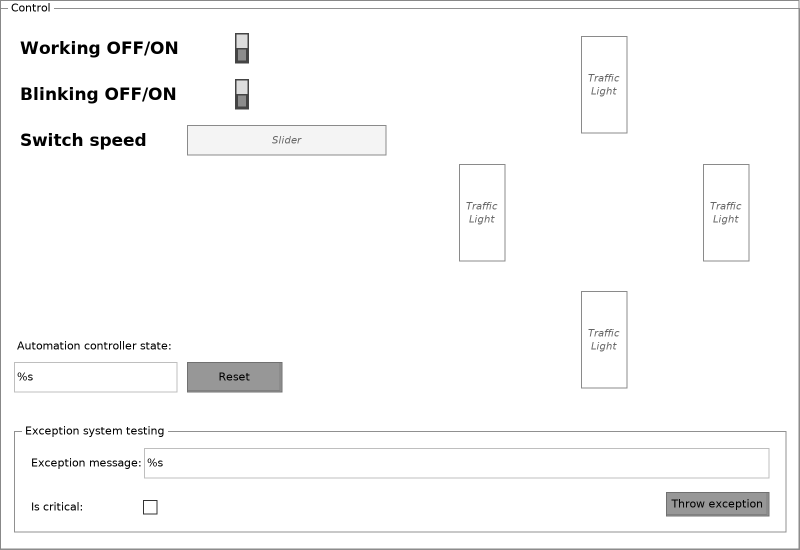
VISUALIZATION Intersection  // 800x550
    GroupBox (0,0 800x550), "Control"
        Label (17,33 166x30), "Working OFF/ON"
        Label (17,79 166x30), "Blinking OFF/ON"
        Rectangle (543,32 120x360), angle 90
        Line (486,126)
        Rectangle (543,24 120x376)
        Frame (581,36 46x97)
            shows TrafficLight(Red := Terminals.DO_2.Channel_4, Yellow := Terminals.DO_2.Channel_5, Green := Terminals.DO_2.Channel_6)
        Frame (581,291 46x97)
            shows TrafficLight(Red := Terminals.DO_2.Channel_10, Yellow := Terminals.DO_2.Channel_11, Green := Terminals.DO_2.Channel_12)
        Frame (703,164 46x97)
            shows TrafficLight(Red := Terminals.DO_2.Channel_7, Yellow := Terminals.DO_2.Channel_8, Green := Terminals.DO_2.Channel_9)
        Frame (459,164 46x97)
            shows TrafficLight(Red := Terminals.DO_2.Channel_1, Yellow := Terminals.DO_2.Channel_2, Green := Terminals.DO_2.Channel_3)
        DipSwitch (202,33 80x30), variable: Terminals.DI_1.Channel_1, behaviour: TOGGLE, style: Switch-DipSwitch-Gray
        DipSwitch (202,79 80x30), variable: Terminals.DI_1.Channel_2, behaviour: TOGGLE, style: Switch-DipSwitch-Gray
        Textfield (14,362 163x30), "%s", text variable: MAIN.IntersectionController.OperationalStateName, input disabled if: FALSE
        Label (14,331 270x30), "Automation controller state:"
        Slider (187,125 199x30), variable: Terminals.AI_3.Channel_1.Value, scale -32768..32767
        Label (17,125 166x30), "Switch speed"
        GroupBox (14,423 772x109), "Exception system testing"
            Label (14,25 116x30), "Exception message:"
            Textfield (130,25 625x30), "%s", text variable: MAIN.IntersectionController.TestExceptionMessage, input disabled if: FALSE
                OnMouseClick: write the text variable via Default
            Button (652,69 103x24), "Throw exception"
                OnMouseClick: execute { MAIN.IntersectionController.ThrowTestExceptionRequest := TRUE; }
            Label (14,68 110x30)
            Label (14,69 110x30), "Is critical:"
            Checkbox (127,69 28x30), variable: MAIN.IntersectionController.IsTestExceptionCritical
        Button (187,362 95x30), "Reset"
            OnMouseClick: execute { MAIN.IntersectionController.ResetRequest := TRUE; }
END_VISUALIZATION

(* stored: Version 1.1.0.1
   Visu Intersection: Id {3f36056b-e97d-47c4-837d-733890435638} *)
